TEXTLIST CommandList
  1 = 'Reset'
  2 = 'Power'
  3 = 'Read Status'
  4 = 'Read Axis Error'
  5 = 'Read Parameter'
  6 = 'Read Bool Parameter'
  7 = 'Write Parameter'
  8 = 'Write Bool Parameter'
  9 = 'Read Digital Input *'
  10 = 'Read Digital Output*'
  11 = 'Write Digital Output*'
  12 = 'Read Actual Position'
  13 = 'Read Actual Velocity'
  14 = 'Read Actual Torque*'
  15 = 'Read Axis Info*'
  16 = 'Read Motion State *'
  17 = 'Set Position'
  18 = 'Set Override'
  19 = 'Touch Probe'
  20 = 'Digital Cam Switch *'
  21 = 'Abort Trigger'
  22 = 'Abort Superposition'
  23 = 'Cam Table Select'
  24 = 'Home'
  25 = 'Jog'
  26 = 'Stop'
  27 = 'Halt'
  28 = 'Move Absolute'
  29 = 'Move Relative'
  30 = 'Move Additive'
  31 = 'Move Superimposed'
  32 = 'Move Velocity'
  33 = 'Move Continuous Absolute'
  34 = 'Move Continuous Relative'
  35 = 'Move Modulo'
  36 = 'Torque Control *'
  37 = 'Position Profile *'
  38 = 'Velocity Profile *'
  39 = 'Acceleration Profile *'
  40 = 'Gear In'
  41 = 'Gear In Dynamic'
  42 = 'Gear In Multi-Master'
  43 = 'Gear Out'
  44 = 'Halt Phasing'
  45 = 'Phasing Absolute'
  46 = 'Phasing Relative'
  47 = 'Cam In'
  48 = 'Cam Out'
  49 = 'Cam Scaling'
  50 = 'Cam Add'
  51 = 'Cam Exchange'
  52 = 'Cam In V2'
  53 = 'Cam Remove'
  54 = 'Cam Scaling V2'
   = ''
END_TEXTLIST

(* stored: Version 1.1.0.1, ProductVersion 3.1.4022.12
   TextList CommandList: Id {85c9ae21-2fcb-40d3-8ece-7d9f0cadc9e8} *)
